# EPICS autosave request: ttiCPX/ttiCPX_channel_settings.req
$(P):$(CHAN):CURRENT
$(P):$(CHAN):OUTPUT
$(P):$(CHAN):VOLTAGE
